INTERFACE ITcoObject EXTENDS __SYSTEM.IQueryInterface

{attribute 'hide'}
PROPERTY Context : ITcoContext
GET
END_GET
END_PROPERTY

PROPERTY Identity : ULINT
GET
END_GET
END_PROPERTY

END_INTERFACE

(* stored: Version 1.1.0.1
   Itf ITcoObject: Id {23caff12-ced5-4482-b750-087e4e453b79}
   Property Context: Id {02fcb32b-7113-4674-b89a-f6974d243c58}
   Get Get: Id {4408d60f-27dd-4547-b759-df6566bc3f65}
   Property Identity: Id {e24e6aab-d37c-4251-a2f9-c1cd4070513a}
   Get Get: Id {4f5fda5b-34c0-4185-ba6e-77c2c887aef7} *)
